# EPICS substitutions: CSTestBench/iocs/BL99I-LCH-IOC-01/BL99I-LCH-IOC-01App/Db/BL99I-LCH-IOC-01_expanded.substitutions
# This file was automatically generated on Mon 20 Apr 2020 07:42:15 BST from
# source: /home/jjc62351/work/builderTestBench/CSTestBench/etc/makeIocs/BL99I-LCH-IOC-01.xml
#
# *** Please do not edit this file: edit the source file instead. ***
#

# Macros:
#  PORT      The asyn port for the pmac controller
#  P         PV Prefix
#  NAXES     Number of axes
#  TIMEOUT   Timeout for controller communication
#  FEEDRATE  feedrate below which we go into error
#  CSG0      Name for Coordinate System Group 0
#  CSG1      Name for Coordinate System Group 1
#  CSG2      Name for Coordinate System Group 2
#  CSG3      Name for Coordinate System Group 3
#  CSG4      Name for Coordinate System Group 4
#  CSG5      Name for Coordinate System Group 5
#  CSG6      Name for Coordinate System Group 6
#  CSG7      Name for Coordinate System Group 7
file $(PMAC)/db/pmacController.template
{
pattern { PORT, P, NAXES, TIMEOUT, FEEDRATE, CSG0, CSG1, CSG2, CSG3, CSG4, CSG5, CSG6, CSG7 }
    { "BRICK11", "BL99I-MO-STEP-11", "8", "4", "100", "", "", "", "", "", "", "", "" }
}

# Macros:
#  PORT  The asyn port for the pmac controller
#  P     PV Prefix
file $(PMAC)/db/pmacStatus.template
{
pattern { PORT, P }
    { "BRICK11", "BL99I-MO-STEP-11" }
}

# Macros:
#  PMAC  Pmac/Geobrick name
#  AXIS  Axis number
#  PORT  Asyn port
file $(PMAC)/db/pmacStatusAxis.template
{
pattern { PMAC, AXIS, PORT }
    { "BL99I-MO-STEP-11", "1", "BRICK11" }
    { "BL99I-MO-STEP-11", "2", "BRICK11" }
    { "BL99I-MO-STEP-11", "3", "BRICK11" }
    { "BL99I-MO-STEP-11", "4", "BRICK11" }
    { "BL99I-MO-STEP-11", "5", "BRICK11" }
    { "BL99I-MO-STEP-11", "6", "BRICK11" }
    { "BL99I-MO-STEP-11", "7", "BRICK11" }
    { "BL99I-MO-STEP-11", "8", "BRICK11" }
}

# Macros:
#  P                Device Prefix
#  M                Device Suffix
#  PORT             Delta tau motor controller
#  ADDR             Address on controller
#  DESC             Description, displayed on EDM screen
#  MRES             Motor Step Size (EGU)
#  VELO             Velocity (EGU/s)
#  PREC             Display Precision
#  EGU              Engineering Units
#  TWV              Tweak Step Size (EGU)
#  DTYP             DTYP of record
#  DIR              User Direction
#  VBAS             Base Velocity (EGU/s)
#  VMAX             Max Velocity (EGU/s), defaults to VELO
#  ACCL             Seconds to Velocity
#  BDST             BL Distance (EGU)
#  BVEL             BL Velocity (EGU/s)
#  BACC             BL Seconds to Veloc.
#  DHLM             Dial High Limit
#  DLLM             Dial Low Limit
#  HLM              User High Limit
#  LLM              User Low Limit
#  HLSV             HW Lim. Violation Svr
#  INIT             Startup commands
#  SREV             Steps per Revolution
#  RRES             Readback Step Size (EGU)
#  ERES             Encoder Step Size (EGU)
#  JAR              Jog Acceleration (EGU/s^2)
#  UEIP             Use Encoder If Present
#  URIP             Use RDBL If Present
#  RDBL             Readback Location, set URIP = 1 if you specify this
#  RLNK             Readback output link
#  RTRY             Max retry count
#  DLY              Readback settle time (s)
#  OFF              User Offset (EGU)
#  RDBD             Retry Deadband (EGU)
#  FOFF             Freeze Offset, 0=variable, 1=frozen
#  ADEL             Alarm monitor deadband (EGU)
#  NTM              New Target Monitor, only set to 0 for soft motors
#  FEHIGH           HIGH limit for following error
#  FEHIHI           HIHI limit for following error
#  FEHHSV           HIHI alarm severity for following error
#  FEHSV            HIGH alarm severity for following error
#  SCALE            Scale factor, if pmacSetAxisScale is used this should be set
#  HOMEVIS          If 1 then home is visible on the gui
#  HOMEVISSTR       If HOMEVIS=0, then display this text on the gui instead
#  name             Object name and gui association name
#  alh              Set this to alh to add the motor to the alarm handler and send emails,
#  gda_name         Name to export this as to GDA
#  gda_desc         Description to export this as to GDA
#  SPORT            Delta tau motor controller comms port
#  HOME             Prefix for autohome instance. Defaults to $(P). If unspecified,
#  ALLOW_HOMED_SET  Set to a blank to allow this axis to have its homed
file $(PMAC)/db/dls_pmac_asyn_motor.template
{
pattern { P, M, PORT, ADDR, DESC, MRES, VELO, PREC, EGU, TWV, DTYP, DIR, VBAS, VMAX, ACCL, BDST, BVEL, BACC, DHLM, DLLM, HLM, LLM, HLSV, INIT, SREV, RRES, ERES, JAR, UEIP, URIP, RDBL, RLNK, RTRY, DLY, OFF, RDBD, FOFF, ADEL, NTM, FEHIGH, FEHIHI, FEHHSV, FEHSV, SCALE, HOMEVIS, HOMEVISSTR, name, alh, gda_name, gda_desc, SPORT, HOME, PMAC, ALLOW_HOMED_SET }
    { "BL99I-AL-SLITS-04", ":XCENTRE", "BRICK11", "1", "Slits S4 X Centre", "0.01", "1", "6", "mm", "0.1", "asynMotor", "0", "0", "$(VELO)", "0.5", "0", "0", "", "13", "-13", "", "", "MAJOR", "", "1000", "", "", "", "0", "0", "", "", "0", "0", "0", "", "0", "0", "1", "0", "0", "NO_ALARM", "NO_ALARM", "1", "1", "Use motor summary screen", "S4.XCEN", "None", "", "$(DESC)", "BRICK11Port", "$(P)", "BL99I-MO-STEP-11", "#" }
    { "BL99I-AL-SLITS-04", ":XSIZE", "BRICK11", "2", "Slits S4 X Size", "0.01", "1", "6", "mm", "0.1", "asynMotor", "0", "0", "$(VELO)", "0.5", "0", "0", "", "13", "-13", "", "", "MAJOR", "", "1000", "", "", "", "0", "0", "", "", "0", "0", "0", "", "0", "0", "1", "0", "0", "NO_ALARM", "NO_ALARM", "1", "1", "Use motor summary screen", "S4.XSIZE", "None", "", "$(DESC)", "BRICK11Port", "$(P)", "BL99I-MO-STEP-11", "#" }
    { "BL99I-AL-SLITS-04", ":YCENTRE", "BRICK11", "3", "Slits S4 Y Centre", "0.01", "1", "6", "mm", "0.1", "asynMotor", "0", "0", "$(VELO)", "0.5", "0", "0", "", "13", "-13", "", "", "MAJOR", "", "1000", "", "", "", "0", "0", "", "", "0", "0", "0", "", "0", "0", "1", "0", "0", "NO_ALARM", "NO_ALARM", "1", "1", "Use motor summary screen", "S4.YCEN", "None", "", "$(DESC)", "BRICK11Port", "$(P)", "BL99I-MO-STEP-11", "#" }
}

# Macros:
#  motor    Device prefix
#  PRE_POS  Position to move to before move
#  name     Gui element
#  DESC     Template argument
file $(BL11K)/db/benderMove.template
{
pattern { motor, PRE_POS, name, DESC }
    { "BL99I-AL-SLITS-04:XCENTRE", "1", "BMOV", "" }
}
